Staubli VAL3: saveHomeBox.dtx

mdesc mNomSpeed
public num nBoxType = 1
